
FUNCTION CB_max_time : TIME

TITLE = ' Search for the greater variable '
VERSION : '1.0'
AUTHOR  : CB
NAME    : maxTime
FAMILY  : TNI

VAR_INPUT
    IN0 : TIME;
    IN1 : TIME;
END_VAR

BEGIN

    CB_max_time := MAX(IN1 := IN0, IN2 := IN1);

END_FUNCTION
